// TIA Portal project "Sort Boxes Based on weight" (V19)

(* hardware
DEVICE "S7-1200 station_1"  S7-1200 Station
   slot 0: "Rack_0"  S7-1200 Rack  Rack  V1.0
   slot 1: "PLC_1"  CPU 1211C AC/DC/Rly  6ES7 211-1BE40-0XB0  V4.6
DEVICE "HMI_1"  KTP400 Basic PN
   slot 0: "HMI_1"  KTP400 Basic PN  6AV2 123-2DB03-0AX0  17.0.0.0
   slot 1: "HMI_RT_1"  KTP400 Basic PN  6AV2 123-2DB03-0AX0  17.0.0.0
   slot 5: "HMI_1.IE_CP_1"  PROFINET Interface  17.0.0.0
      slot 1: "PROFINET Interface_1"  PROFINET Interface
         slot 1: "Port_1"  Port
*)

// ===== PLC "PLC_1"  CPU 1211C AC/DC/Rly =====

VAR_GLOBAL   // PLC tag table "Default tag table"
   "START PB" AT %I0.0 : Bool;
   "Reset Button 0" AT %I0.1 : Bool;
   "Stop sensor" AT %I0.2 : Bool;
   "EXIT SENSOR LEFT" AT %I0.3 : Bool;
   "EXIT SENSOR MIDDLE" AT %I0.4 : Bool;
   "EXIT SENSOR RIGHT" AT %I0.5 : Bool;
   "MAIN CONVEYOR" AT %Q0.0 : Bool;
   "Conveyor Scale 0 (+)" AT %Q0.1 : Bool;
   "SORT FORWARD" AT %Q0.2 : Bool;
   "SORT LEFT" AT %Q0.3 : Bool;
   "SORT RIGHT" AT %Q0.4 : Bool;
   "LEFT CONVEYOR" AT %Q0.5 : Bool;
   "MIDDLE CONVEYOR" AT %Q0.6 : Bool;
   "RIGHT CONVEYOR" AT %Q0.7 : Bool;
   "Conveyor Scale 0 Weight (V)" AT %ID30 : Real;
   "8KG BOX COUNTER" AT %QD30 : Real;
   "10KG BOX COUNTER" AT %QD34 : Real;
   "15KG BOX COUNTER" AT %QD38 : Real;
   "Tag_1" AT %Q2.0 : Bool;
   "Tag_2" AT %Q3.0 : Bool;
   "Tag_3" AT %MD0 : Real;
   "Tag_4" AT %MD2 : DWord;
   "Tag_5" AT %M0.0 : Bool;
   "Tag_6" AT %MD38 : DWord;
   "Tag_7" AT %MD4 : DWord;
   "START INDICATOR" AT %M1.4 : Bool;
   "STOP INDICATOR" AT %M1.6 : Bool;
   "Tag_8" AT %M0.2 : Bool;
   "HMI_START_PB" AT %M10.0 : Bool;
   "HMI_STOP_PB" AT %M10.2 : Bool;
   "Tag_9" AT %M10.4 : Bool;
END_VAR

// folder: System blocks/Program resources

DATA_BLOCK "IEC_Timer_0_DB"   // DB1
{ S7_Optimized_Access := 'TRUE' }
AUTHOR : Simatic
FAMILY : IEC
NAME : IEC_TMR
VERSION : 1.0
// stored: InstanceOfName IEC_TIMER
"IEC_TIMER"
BEGIN
END_DATA_BLOCK

DATA_BLOCK "IEC_Timer_0_DB_3"   // DB2
{ S7_Optimized_Access := 'TRUE' }
AUTHOR : Simatic
FAMILY : IEC
NAME : IEC_TMR
VERSION : 1.0
// stored: InstanceOfName IEC_TIMER
"IEC_TIMER"
BEGIN
END_DATA_BLOCK

DATA_BLOCK "IEC_Counter_0_DB"   // DB3
{ S7_Optimized_Access := 'TRUE' }
AUTHOR : Simatic
FAMILY : IEC
NAME : CNTR
VERSION : 1.0
// stored: InstanceOfName IEC_COUNTER
"IEC_COUNTER"
BEGIN
END_DATA_BLOCK

DATA_BLOCK "IEC_Counter_0_DB_1"   // DB4
{ S7_Optimized_Access := 'TRUE' }
AUTHOR : Simatic
FAMILY : IEC
NAME : CNTR
VERSION : 1.0
// stored: InstanceOfName IEC_COUNTER
"IEC_COUNTER"
BEGIN
END_DATA_BLOCK

DATA_BLOCK "IEC_Counter_0_DB_2"   // DB5
{ S7_Optimized_Access := 'TRUE' }
AUTHOR : Simatic
FAMILY : IEC
NAME : CNTR
VERSION : 1.0
// stored: InstanceOfName IEC_COUNTER
"IEC_COUNTER"
BEGIN
END_DATA_BLOCK

// folder: (top level)

FUNCTION "MHJ-PLC-Lab-Function-S71200" : Void   // FC9000, SCL
{ S7_Optimized_Access := 'TRUE' }
VERSION : 0.1
   VAR_TEMP
      rdTimeReturn : Int;
      outputTime : DTL;
      SyncVal : Byte;
      forVal : Int;
      forVal_2 : Int;
      Value : Byte;
   END_VAR
   VAR CONSTANT
      CompVal : Byte := 16#34;
      Value_01 : Byte := 16#11;
      Value_01_DW : DWord := 16#A165_D992;
      Value_02_DW : DWord := 16#58BE_4401;
   END_VAR
BEGIN

   #Value:=PEEK(area := 16#82,
        dbNumber := 0,
        byteOffset := 511);
   #Value := #Value + 1;

   POKE(area := 16#82,
        dbNumber := 0,
        byteOffset := 511,
        value := #Value);

   POKE(area:=16#81,
        dbNumber:=0,
        byteOffset:=1016,
        value:=#Value_01_DW);
   POKE(area := 16#81,
        dbNumber := 0,
        byteOffset := 1020,
        value := #Value_02_DW);

   POKE(area := 16#81,
        dbNumber := 0,
        byteOffset := 511,
        value := B#16#00);

   FOR #forVal := 0 TO 120 DO
       FOR #forVal_2:=0 TO 10 DO
           #rdTimeReturn:=RD_SYS_T(#outputTime);
           #rdTimeReturn := WR_SYS_T(#outputTime);
           #rdTimeReturn := RD_SYS_T(#outputTime);
           #rdTimeReturn := WR_SYS_T(#outputTime);
       END_FOR;
       #SyncVal:= PEEK(area := 16#81,
                      dbNumber := 0,
                      byteOffset := 511);
       IF #SyncVal = #CompVal THEN
          GOTO M_1;
       END_IF;
   END_FOR;
   RETURN;

   M_1:
   POKE(area := 16#81,
        dbNumber := 0,
        byteOffset := 511,
        value := B#16#0);
END_FUNCTION

ORGANIZATION_BLOCK "Main"   // OB1, LAD, ProgramCycle
TITLE = "Main Program Sweep (Cycle)"
{ S7_Optimized_Access := 'TRUE' }
VERSION : 0.1
   VAR_INPUT
      Initial_Call : Bool;   // Initial call of this OB
      Remanence : Bool;   // =True, if remanent data are available
   END_VAR
   VAR_TEMP   // added for the SCL form of the ladder/FBD networks
      _w1 : Bool;
      _w2 : Bool;
   END_VAR
BEGIN

REGION Network 1
   // FACTORYIO
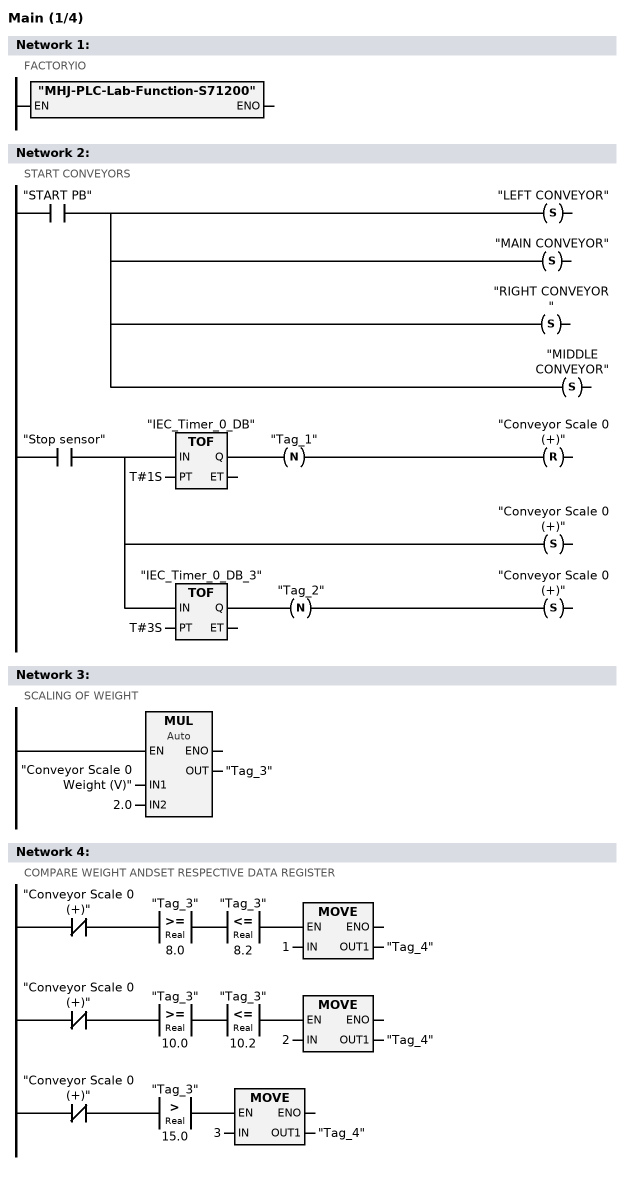
   RUNG wire#powerrail
      "MHJ-PLC-Lab-Function-S71200"()
   END_RUNG
   // the same network as SCL:
   "MHJ-PLC-Lab-Function-S71200"();
END_REGION

REGION Network 2
   // START CONVEYORS
   IF "START PB" THEN
       "LEFT CONVEYOR" := TRUE;
       "MAIN CONVEYOR" := TRUE;
       "RIGHT CONVEYOR" := TRUE;
       "MIDDLE CONVEYOR" := TRUE;
   END_IF;
   "IEC_Timer_0_DB".TOF(IN := "Stop sensor", PT := T#1S);
   #_w1 := NOT "IEC_Timer_0_DB".Q AND "Tag_1";   // falling edge
   "Tag_1" := "IEC_Timer_0_DB".Q;
   IF #_w1 THEN "Conveyor Scale 0 (+)" := FALSE; END_IF;
   IF "Stop sensor" THEN "Conveyor Scale 0 (+)" := TRUE; END_IF;
   "IEC_Timer_0_DB_3".TOF(IN := "Stop sensor", PT := T#3S);
   #_w2 := NOT "IEC_Timer_0_DB_3".Q AND "Tag_2";   // falling edge
   "Tag_2" := "IEC_Timer_0_DB_3".Q;
   IF #_w2 THEN "Conveyor Scale 0 (+)" := TRUE; END_IF;
END_REGION

REGION Network 3
   // SCALING OF WEIGHT
   RUNG wire#powerrail
      Mul(in1 := "Conveyor Scale 0 Weight (V)", in2 := 2.0, out => "Tag_3")
   END_RUNG
   // the same network as SCL:
   "Tag_3" := "Conveyor Scale 0 Weight (V)" * 2.0;
END_REGION

REGION Network 4
   // COMPARE WEIGHT ANDSET RESPECTIVE DATA REGISTER
   RUNG wire#powerrail
      I_Contact( "Conveyor Scale 0 (+)" )
      { S7_Templates := "SrcType := Real" } GE_Contact(in1 := "Tag_3", in2 := 8.0)
      { S7_Templates := "SrcType := Real" } LE_Contact(in1 := "Tag_3", in2 := 8.2)
      Move(in := 1, out1 => "Tag_4")
   END_RUNG
   RUNG wire#powerrail
      I_Contact( "Conveyor Scale 0 (+)" )
      { S7_Templates := "SrcType := Real" } GE_Contact(in1 := "Tag_3", in2 := 10.0)
      { S7_Templates := "SrcType := Real" } LE_Contact(in1 := "Tag_3", in2 := 10.2)
      Move(in := 2, out1 => "Tag_4")
   END_RUNG
   RUNG wire#powerrail
      I_Contact( "Conveyor Scale 0 (+)" )
      { S7_Templates := "SrcType := Real" } GT_Contact(in1 := "Tag_3", in2 := 15.0)
      Move(in := 3, out1 => "Tag_4")
   END_RUNG
   // the same network as SCL:
   IF NOT "Conveyor Scale 0 (+)" AND ("Tag_3" >= 8.0) AND ("Tag_3" <= 8.2) THEN "Tag_4" := 1; END_IF;
   IF NOT "Conveyor Scale 0 (+)" AND ("Tag_3" >= 10.0) AND ("Tag_3" <= 10.2) THEN "Tag_4" := 2; END_IF;
   IF NOT "Conveyor Scale 0 (+)" AND ("Tag_3" > 15.0) THEN "Tag_4" := 3; END_IF;
END_REGION

REGION Network 5
   // SORT LEFT BOX
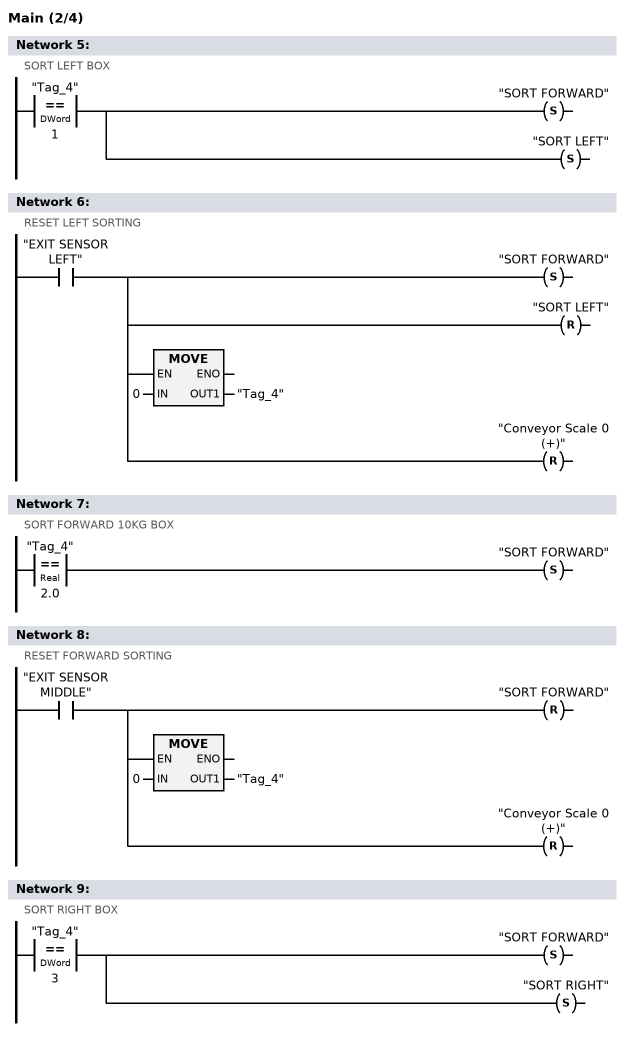
   RUNG wire#powerrail
      { S7_Templates := "SrcType := DWord" } EQ_Contact(in1 := "Tag_4", in2 := 1)
      wire#w1
      S_Coil( "SORT FORWARD" )
   END_RUNG
   RUNG wire#w1
      S_Coil( "SORT LEFT" )
   END_RUNG
   // the same network as SCL:
   IF "Tag_4" = 1 THEN
       "SORT FORWARD" := TRUE;
       "SORT LEFT" := TRUE;
   END_IF;
END_REGION

REGION Network 6
   // RESET LEFT SORTING
   RUNG wire#powerrail
      Contact( "EXIT SENSOR LEFT" )
      wire#w1
      S_Coil( "SORT FORWARD" )
   END_RUNG
   RUNG wire#w1
      R_Coil( "SORT LEFT" )
   END_RUNG
   RUNG wire#w1
      Move(in := 0, out1 => "Tag_4")
   END_RUNG
   RUNG wire#w1
      R_Coil( "Conveyor Scale 0 (+)" )
   END_RUNG
   // the same network as SCL:
   IF "EXIT SENSOR LEFT" THEN
       "SORT FORWARD" := TRUE;
       "SORT LEFT" := FALSE;
       "Tag_4" := 0;
       "Conveyor Scale 0 (+)" := FALSE;
   END_IF;
END_REGION

REGION Network 7
   // SORT FORWARD 10KG BOX
   RUNG wire#powerrail
      { S7_Templates := "SrcType := Real" } EQ_Contact(in1 := "Tag_4", in2 := 2.0)
      S_Coil( "SORT FORWARD" )
   END_RUNG
   // the same network as SCL:
   IF "Tag_4" = 2.0 THEN "SORT FORWARD" := TRUE; END_IF;
END_REGION

REGION Network 8
   // RESET FORWARD SORTING
   RUNG wire#powerrail
      Contact( "EXIT SENSOR MIDDLE" )
      wire#w1
      R_Coil( "SORT FORWARD" )
   END_RUNG
   RUNG wire#w1
      Move(in := 0, out1 => "Tag_4")
   END_RUNG
   RUNG wire#w1
      R_Coil( "Conveyor Scale 0 (+)" )
   END_RUNG
   // the same network as SCL:
   IF "EXIT SENSOR MIDDLE" THEN
       "SORT FORWARD" := FALSE;
       "Tag_4" := 0;
       "Conveyor Scale 0 (+)" := FALSE;
   END_IF;
END_REGION

REGION Network 9
   // SORT RIGHT BOX
   RUNG wire#powerrail
      { S7_Templates := "SrcType := DWord" } EQ_Contact(in1 := "Tag_4", in2 := 3)
      wire#w1
      S_Coil( "SORT FORWARD" )
   END_RUNG
   RUNG wire#w1
      S_Coil( "SORT RIGHT" )
   END_RUNG
   // the same network as SCL:
   IF "Tag_4" = 3 THEN
       "SORT FORWARD" := TRUE;
       "SORT RIGHT" := TRUE;
   END_IF;
END_REGION

REGION Network 10
   // RESET RIGHT SORTING
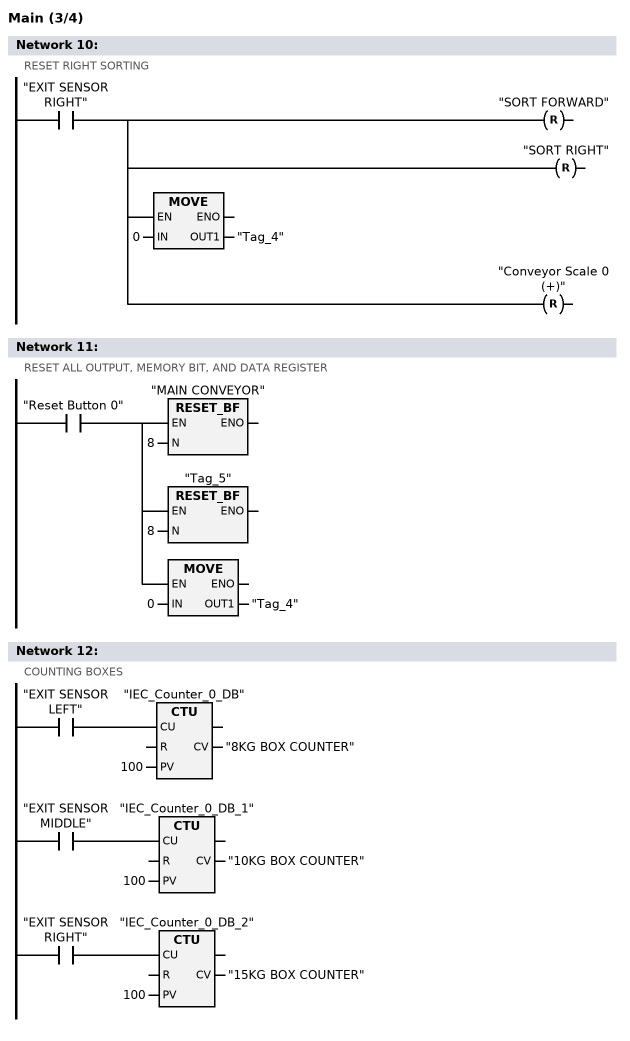
   RUNG wire#powerrail
      Contact( "EXIT SENSOR RIGHT" )
      wire#w1
      R_Coil( "SORT FORWARD" )
   END_RUNG
   RUNG wire#w1
      R_Coil( "SORT RIGHT" )
   END_RUNG
   RUNG wire#w1
      Move(in := 0, out1 => "Tag_4")
   END_RUNG
   RUNG wire#w1
      R_Coil( "Conveyor Scale 0 (+)" )
   END_RUNG
   // the same network as SCL:
   IF "EXIT SENSOR RIGHT" THEN
       "SORT FORWARD" := FALSE;
       "SORT RIGHT" := FALSE;
       "Tag_4" := 0;
       "Conveyor Scale 0 (+)" := FALSE;
   END_IF;
END_REGION

REGION Network 11
   // RESET ALL OUTPUT, MEMORY BIT, AND DATA REGISTER
   // no SCL statement known for RBitfield: written as a call
   #_w1 := "Reset Button 0";
   IF #_w1 THEN
       RESET_BF(operand := "MAIN CONVEYOR", n := 8);
       RESET_BF(operand := "Tag_5", n := 8);
       "Tag_4" := 0;
   END_IF;
END_REGION

REGION Network 12
   // COUNTING BOXES
   "IEC_Counter_0_DB".CTU(CU := "EXIT SENSOR LEFT", PV := 100, CV => "8KG BOX COUNTER");
   "IEC_Counter_0_DB_1".CTU(CU := "EXIT SENSOR MIDDLE", PV := 100, CV => "10KG BOX COUNTER");
   "IEC_Counter_0_DB_2".CTU(CU := "EXIT SENSOR RIGHT", PV := 100, CV => "15KG BOX COUNTER");
END_REGION

REGION Network 13
   // HMI INDICATORS
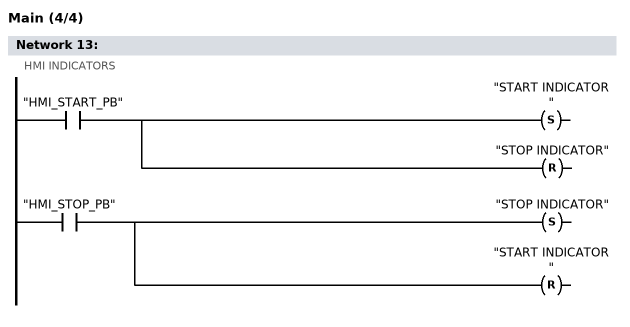
   RUNG wire#powerrail
      Contact( "HMI_START_PB" )
      wire#w1
      S_Coil( "START INDICATOR" )
   END_RUNG
   RUNG wire#w1
      R_Coil( "STOP INDICATOR" )
   END_RUNG
   RUNG wire#powerrail
      Contact( "HMI_STOP_PB" )
      wire#w2
      S_Coil( "STOP INDICATOR" )
   END_RUNG
   RUNG wire#w2
      R_Coil( "START INDICATOR" )
   END_RUNG
   // the same network as SCL:
   IF "HMI_START_PB" THEN
       "START INDICATOR" := TRUE;
       "STOP INDICATOR" := FALSE;
   END_IF;
   IF "HMI_STOP_PB" THEN
       "STOP INDICATOR" := TRUE;
       "START INDICATOR" := FALSE;
   END_IF;
END_REGION
END_ORGANIZATION_BLOCK

(* ===== HMI "HMI_RT_1" =====
system functions are stored by id; their names below are inferred from use
connection "HMI_Connection_1": ETHERNET, SMART_S7_1200_OMS

HMI tags "Default tag table"
   "START PB" : Bool = PLC "START PB" AT %I0.0, 100 ms
   "Reset Button 0" : Bool = PLC "Reset Button 0" AT %I0.1, 1 s
   "IEC_Timer_0_DB_3_Q" : Bool = PLC IEC_Timer_0_DB_3.Q, 1 s
   "8KG BOX COUNTER" : Real = PLC "8KG BOX COUNTER" AT %QD30, 1 s
   "10KG BOX COUNTER" : Real = PLC "10KG BOX COUNTER" AT %QD34, 1 s
   "15KG BOX COUNTER" : Real = PLC "15KG BOX COUNTER" AT %QD38, 1 s
   "START INDICATOR" : Bool = PLC "START INDICATOR" AT %M1.4, 100 ms
   "STOP INDICATOR" : Bool = PLC "STOP INDICATOR" AT %M1.6, 100 ms
   "HMI_START_PB" : Bool = PLC HMI_START_PB AT %M10.0, 1 s
   "HMI_STOP_PB" : Bool = PLC HMI_STOP_PB AT %M10.2, 1 s

Template "Template_1" 480x272
   Button "Exit" at 388,227 size 63x44; TextOff 'Exit'; PictureOff "ExitRuntime_KTP400_Basic_PN_TR"; PictureOn "ExitRuntime_KTP400_Basic_PN_TR"
      on Release: StopRuntime(0)
   Button "Template_Button" at 268,227 size 63x44; TextOff 'Text'
   Button "Template_Button_1" at 148,227 size 63x44; TextOff 'Text'
   Button "Start screen" at 28,227 size 63x44; TextOff 'Start screen'; PictureOff "NavigateHome_KTP400_Basic_PN_TR"; PictureOn "NavigateHome_KTP400_Basic_PN_TR"
      on Release: ActivateScreen("Root screen", 0)

screen "Root screen" 480x272, template "Template_1"
   Button "Button_1" at 293,51 size 96x32; TextOff 'START'
      on Press: SetBit("START PB")
      on Release: SetBit("HMI_START_PB"); InvertBit("HMI_STOP_PB")
   Button "Button_2" at 294,104 size 96x32; TextOff 'STOP'
      on Press: SetBit("Reset Button 0")
      on Release: SetBit("HMI_STOP_PB"); InvertBit("HMI_START_PB")
   Circle "Circle_1" at 417,51 size 32x32
      Appearance <- "START INDICATOR"
   Circle "Circle_2" at 417,103 size 32x32
      Appearance <- "STOP INDICATOR"
   IOField "I/O field_1" at 63,43 size 96x32; FormatPattern s999999999.999
      ProcessValue <- "8KG BOX COUNTER"
   TextField "Text field_1" at 63,19 size 74x20; Text '8KG BOXES'
   IOField "I/O field_2" at 63,105 size 96x32; FormatPattern s999999999.999
      ProcessValue <- "10KG BOX COUNTER"
   TextField "Text field_2" at 63,83 size 82x20; Text '10KG BOXES'
   IOField "I/O field_3" at 63,169 size 96x32; FormatPattern s999999999.999
      ProcessValue <- "15KG BOX COUNTER"
   TextField "Text field_3" at 63,149 size 82x20; Text '15KG BOXES'
*)